# EPICS StreamDevice protocol: htscope1/protocols/hts.proto
Terminator = LF;
ExtraInput = Ignore;
ReplyTimeout = 2500;

getIDLE {
	in "waiting %d\r";
}

getRunTime {
    in "%s\r";
}
